// TIA Portal V17 export
// export: Created 2026-01-01T00:00:00, ExportSetting WithDefaults, DisplayName synthetic-fixture, DisplayVersion machine-intelligence-v1.0.0
FUNCTION "FC_Mode" : Void   // FC, SCL
BEGIN

NETWORK
TITLE = 
AutoMode := Auto AND NOT Manual;
END_FUNCTION
